Fanuc TP program (LS listing): FOLGE020.LS

/PROG  FOLGE020
/ATTR
OWNER		= GME;
COMMENT		= "VW336";
PROG_SIZE	= 7468;
CREATE		= DATE 16-09-30  TIME 23:12:18;
MODIFIED	= DATE 23-07-29  TIME 10:10:58;
FILE_NAME	= FOLGE020;
VERSION		= 0;
LINE_COUNT	= 47;
MEMORY_SIZE	= 11772;
PROTECT		= READ_WRITE;
TCD:  STACK_SIZE	= 500,
      TASK_PRIORITY	= 50,
      TIME_SLICE	= 0,
      BUSY_LAMP_OFF	= 0,
      ABORT_REQUEST	= 0,
      PAUSE_REQUEST	= 0;
DEFAULT_GROUP	= 1,1,1,1,*;
CONTROL_CODE	= 00000000 00000000;
/APPL
/MN
   1:  UFRAME_NUM=0 ;
   2:  UTOOL_NUM=1 ;
   3:  PAYLOAD[1] ;
   4:J P[1] 10% CNT0 ACC100 TB   0.00sec,P-SPS    ;
      1:  IF (DO[12]),CALL MAKRO998 ;
      2:  DO[15]=ON ;
      3:  DO[16]=ON ;
      4:  CALL MAKRO000    ;
      5:  WAIT (DI[9])    ;
       ------ ;
   5:  !Liberaciones PLC ;
   6:  !Fresado Estacionario SP1 ;
   7:  !Purgar KL1 ;
   8:J P[2] 100% CNT0 ACC100 TB   0.00sec,P-SPS    ;
      1:  TC_ONLINE (ON) ;
      4:  DO[23]=OFF ;
     32:  !Apagar Posicion base ;
     33:  DO[15]=OFF ;
      2:  !Espera fin de purga en casa ;
      3:  WAIT ((!DI[1534] AND !DI[1535]) OR !F[346] OR DI[15])    ;
      5:  TIMER[1]=RESET ;
      6:  TIMER[1]=START ;
      7:  CALL MAKRO050    ;
      8:  !Lib. Herramientas ;
      9:  DO[80]=ON ;
     10:  DO[79]=ON ;
     11:  DO[78]=OFF ;
     12:  DO[77]=OFF ;
     13:  DO[76]=ON ;
     14:  DO[75]=OFF ;
     15:  DO[74]=OFF ;
     16:  DO[73]=ON ;
     17:  DO[72]=ON ;
     18:  DO[71]=OFF ;
     19:  DO[70]=OFF ;
     20:  DO[69]=OFF ;
     21:  DO[68]=OFF ;
     22:  DO[67]=OFF ;
     23:  !Anticolisiones Robot ;
     24:  DO[41]=ON ;
     25:  DO[42]=ON ;
     26:  DO[43]=ON ;
     27:  DO[44]=ON ;
     28:  DO[53]=ON ;
     29:  DO[54]=ON ;
     30:  DO[55]=ON ;
     31:  DO[56]=ON ;
     34:  !Inicializar Garra ;
     35:  WAIT (M[2])    ;
     36:  F[1]=(ON) ;
     37:  F[2]=(ON) ;
     38:  F[3]=(ON) ;
     39:  F[4]=(ON) ;
     40:  F[5]=(ON) ;
     41:  IF (M[2]),CALL MAKRO342 ;
     42:  CALL MAKRO340    ;
     43:  WAIT (M[31] AND M[33] AND M[35] AND M[37] AND M[39])    ;
     44:  !Fresado SP1 ;
     45:  F[298]=(OFF) ;
     46:  CALL VW_USER(Basic1,EZSP,Nr1,ProgNr=31, , ,S-Punkt=31, ,EIN/AUS=ON) ;
     47:  WAIT    .10(sec) ;
     48:  F[79]=((DI[786] AND !DI[788]) OR (!DI[788] AND DI[130])) ;
     49:  F[78]=(DI[788] AND !F[79]) ;
     50:  GO[2]=(R[197]) ;
     51:  IF (F[78] AND F[79]),CALL MAKRO085 ;
     52:  IF (F[78] OR F[79]),CALL MAKRO084 ;
     53:  WAIT (M[96])    ;
     54:  !Seleccionar Pistola 1 ;
     55:  DO[1521]=ON ;
     56:  DO[1522]=OFF ;
     57:  DO[1523]=OFF ;
     58:  !Confirmacion Pistola 1 ;
     59:  WAIT (DI[1521] AND !DI[1522] AND !DI[1523])    ;
     60:  !Programa ;
     61:  GO[10]=(20) ;
     62:  !Parametro ;
     63:  GO[11]=(1) ;
     64:  WAIT    .10(sec) ;
     65:  !Purgar KL1 ;
     66:  IF (DI[1534] OR DI[163]),CALL MAKRO183 ;
     67:  WAIT (DI[23])    ;
     68:  DO[23]=ON ;
     69:  TC_ONLINE (M[2] AND M[30] AND M[31] AND M[33] AND M[35] AND M[37] AND M[39] AND M[95] AND M[96]) ;
       ------ ;
   9:  !Llamar a UP021 ;
  10:  !Tomar de la Estacion ST1350 ;
  11:  CALL UP021    ;
  12:  UFRAME_NUM=0 ;
  13:  UTOOL_NUM=1 ;
  14:J P[3] 100% CNT0 ACC100 TB    .10sec,P-SPS    ;
      1:  TC_ONLINE (ON) ;
      2:  DO[23]=OFF ;
      3:  WAIT (DI[23])    ;
      4:  DO[23]=ON ;
      5:  TC_ONLINE (M[3] AND M[30] AND M[31] AND M[34] AND M[35] AND M[37] AND M[39] AND M[95] AND M[96]) ;
       ------ ;
  15:  !Llamar a UP022 ;
  16:  !Tomar de la Estacion ST1360 ;
  17:  CALL UP022    ;
  18:  UFRAME_NUM=0 ;
  19:  UTOOL_NUM=1 ;
  20:J P[4] 100% CNT0 ACC100 TB    .10sec,P-SPS    ;
      1:  TC_ONLINE (ON) ;
      2:  DO[23]=OFF ;
      3:  WAIT (DI[23])    ;
      4:  DO[23]=ON ;
      5:  TC_ONLINE (M[1] AND M[30] AND M[31] AND M[34] AND M[36] AND M[38] AND M[39] AND M[95] AND M[96]) ;
       ------ ;
  21:  !Llamar a UP023 ;
  22:  !Soldadura ;
  23:  CALL UP023    ;
  24:  UFRAME_NUM=0 ;
  25:  UTOOL_NUM=1 ;
  26:J P[5] 100% CNT0 ACC100 TB    .10sec,P-SPS    ;
      1:  TC_ONLINE (ON) ;
      2:  DO[23]=OFF ;
      3:  !Fresado EZ1 ;
      4:  F[298]=(OFF) ;
      5:  CALL VW_USER(Basic1,EZSP,Nr1,ProgNr=31, , ,S-Punkt=31, ,EIN/AUS=ON) ;
      6:  WAIT    .10(sec) ;
      7:  F[79]=((DI[786] AND !DI[788]) OR (!DI[788] AND DI[130])) ;
      8:  F[78]=(DI[788] AND !F[79]) ;
      9:  GO[2]=(R[197]) ;
     10:  IF (F[78] OR F[79]),CALL MAKRO085 ;
     11:  IF (F[78] OR F[79]),CALL MAKRO084 ;
     12:  WAIT (M[96])    ;
     13:  WAIT (DI[23])    ;
     14:  DO[23]=ON ;
     15:  TC_ONLINE (M[1] AND M[30] AND M[31] AND M[34] AND M[36] AND M[38] AND M[39] AND M[95] AND M[96]) ;
       ------ ;
  27:  !Purgar ;
  28:  !UP024 Sello Estacionario ;
  29:  !UP070 Posicion Muestra ;
  30:  LBL[1] ;
  31:J P[6] 100% CNT0 ACC100 TB    .10sec,P-SPS    ;
      1:  TC_ONLINE (ON) ;
      2:  DO[23]=OFF ;
      3:  !Purgar KL1 ;
      4:  IF (DI[1534] OR DI[163]),CALL MAKRO183 ;
      5:  WAIT (DI[23])    ;
      6:  DO[23]=ON ;
      7:  TC_ONLINE (M[1] AND M[30] AND M[31] AND M[34] AND M[36] AND M[38] AND M[39] AND M[95] AND M[96]) ;
       ------ ;
  32:  CALL UP024    ;
  33:  IF (F[343] OR DI[162]),CALL UP070 ;
  34:  IF (F[343]),JMP LBL[1] ;
  35:  UFRAME_NUM=0 ;
  36:  UTOOL_NUM=1 ;
  37:  !En Area de Mantenimiento ;
  38:  !Llamar a UP025 ;
  39:  !Dejar en ST1380 ;
  40:J P[7] 100% CNT0 ACC100 TB    .10sec,P-SPS    ;
      1:  TC_ONLINE (ON) ;
      2:  DO[23]=OFF ;
      3:  LBL[1] ;
      4:  DO[18]=(ON) ;
      5:  WAIT ((DI[73] AND DI[72] AND !DI[60] AND DI[59] AND !DI[58] AND DI[57] AND !DI[18]) OR DI[19])    ;
      6:  IF (DI[19]),JMP LBL[3] ;
      7:  IF (DI[73] AND DI[72] AND !DI[60] AND DI[59] AND !DI[58] AND DI[57]),JMP LBL[2] ;
      8:  LBL[3] ;
      9:  IF (F[78] OR F[79]),CALL MAKRO084 ;
     10:  CALL MAKRO089    ;
     11:  DO[17]=(ON) ;
     12:  GO[19]=(11) ;
     13:  F[281]=(ON) ;
     14:  WAIT (DI[17])    ;
     15:  F[64]=(ON) ;
     16:  F[65]=(OFF) ;
     17:  F[66]=(OFF) ;
     18:  F[67]=(OFF) ;
     19:  LBL[4] ;
     20:  IF (DI[132] AND !DI[133] AND !DI[134] AND !DI[135] AND DI[17]),CALL MAKRO081 ;
     21:  IF (F[85]),JMP LBL[4] ;
     22:  CALL VW_USER(Basic1,EZSP,Nr1 Service,ProgNr=31, , ,S-Punkt=31, ,EIN/AUS=1) ;
     23:  F[79]=((!DI[788] AND DI[130]) OR (DI[786] AND !DI[788])) ;
     24:  F[78]=(DI[788] AND !F[79]) ;
     25:  GO[2]=(R[197]) ;
     26:  IF (F[78] OR F[79]),CALL MAKRO085 ;
     27:  IF (F[78] OR F[79]),CALL MAKRO084 ;
     28:  WAIT (M[96] AND !DI[132])    ;
     29:  DO[17]=(OFF) ;
     30:  GO[19]=(0) ;
     31:  WAIT (!DI[19])    ;
     32:  JMP LBL[1] ;
     33:  LBL[2] ;
     34:  DO[18]=(OFF) ;
     35:  F[281]=(OFF) ;
     36:  WAIT (DI[23])    ;
     37:  DO[23]=ON ;
     38:  TC_ONLINE (M[1] AND M[30] AND M[31] AND M[34] AND M[36] AND M[38] AND M[39] AND M[95] AND M[96]) ;
       ------ ;
  41:  CALL UP025    ;
  42:  UFRAME_NUM=0 ;
  43:  UTOOL_NUM=1 ;
  44:J P[8] 100% CNT0 ACC100 TB    .10sec,P-SPS    ;
      1:  TC_ONLINE (ON) ;
      2:  DO[23]=OFF ;
      3:  F[298]=(OFF) ;
      4:  CALL VW_USER(Basic1,EZSP,Nr1,ProgNr=31, , ,S-Punkt=31, ,EIN/AUS=ON) ;
      5:  WAIT    .10(sec) ;
      6:  F[79]=((DI[786] AND !DI[788]) OR (!DI[788] AND DI[130])) ;
      7:  F[78]=(DI[788] AND !F[79]) ;
      8:  GO[2]=(R[197]) ;
      9:  IF (F[78] AND F[79]),CALL MAKRO085 ;
     10:  IF (F[78] OR F[79]),CALL MAKRO084 ;
     11:  WAIT (M[96])    ;
     12:  WAIT (DI[23])    ;
     13:  DO[23]=ON ;
     14:  TC_ONLINE (M[2] AND M[30] AND M[31] AND M[33] AND M[35] AND M[37] AND M[39] AND M[95] AND M[96]) ;
       ------ ;
  45:  !Fin de Trabajo Total ;
  46:J P[9] 100% CNT0 ACC100 TB    .10sec,P-SPS    ;
      1:  TC_ONLINE (ON) ;
      2:  DO[23]=OFF ;
      3:  CALL MAKRO015    ;
      4:  WAIT (DI[23])    ;
      5:  DO[23]=ON ;
      6:  TC_ONLINE (M[2] AND M[30] AND M[31] AND M[33] AND M[35] AND M[37] AND M[39] AND M[95] AND M[96]) ;
       ------ ;
  47:J P[10] 100% CNT0 ACC100 TB   0.00sec,P-SPS    ;
      1:  TC_ONLINE (ON) ;
      2:  DO[14]=ON ;
      3:  DO[15]=ON ;
      4:  TIMER[1]=STOP ;
      5:  TIMER[2]=(TIMER[1]) ;
      6:  TIMER[2]=STOP ;
       ------ ;
/POS
P[1]{
   GP1:
	UF : 0, UT : 1,		CONFIG : 'N U T, 0, 0, -1',
	X =  1190.730  mm,	Y =  -289.205  mm,	Z =  1231.849  mm,
	W =   -30.000 deg,	P =     0.000 deg,	R =    30.000 deg
   GP2:
	UF : 0, UT : 1,
	J1=   100.000  mm
   GP3:
	UF : 0, UT : 1,
	J1=     0.000  mm
   GP4:
	UF : 0, UT : 1,
	J1=     0.000  mm
};
P[2]{
   GP1:
	UF : 0, UT : 1,		CONFIG : 'N U T, 0, 0, -1',
	X =  1190.730  mm,	Y =  -289.205  mm,	Z =  1231.849  mm,
	W =   -30.000 deg,	P =     0.000 deg,	R =    30.000 deg
   GP2:
	UF : 0, UT : 1,
	J1=   100.000  mm
   GP3:
	UF : 0, UT : 1,
	J1=     0.000  mm
   GP4:
	UF : 0, UT : 1,
	J1=     0.000  mm
};
P[3]{
   GP1:
	UF : 0, UT : 1,		CONFIG : 'N U T, 0, 0, -1',
	X =  1190.730  mm,	Y =  -289.205  mm,	Z =  1231.849  mm,
	W =   -30.000 deg,	P =     0.000 deg,	R =    30.000 deg
   GP2:
	UF : 0, UT : 1,
	J1=   100.000  mm
   GP3:
	UF : 0, UT : 1,
	J1=     0.000  mm
   GP4:
	UF : 0, UT : 1,
	J1=     0.000  mm
};
P[4]{
   GP1:
	UF : 0, UT : 1,		CONFIG : 'N U T, 0, 0, -1',
	X =  1190.730  mm,	Y =  -289.205  mm,	Z =  1231.849  mm,
	W =   -30.000 deg,	P =     0.000 deg,	R =    30.000 deg
   GP2:
	UF : 0, UT : 1,
	J1=   100.000  mm
   GP3:
	UF : 0, UT : 1,
	J1=     0.000  mm
   GP4:
	UF : 0, UT : 1,
	J1=     0.000  mm
};
P[5]{
   GP1:
	UF : 0, UT : 1,		CONFIG : 'N U T, 0, 0, -1',
	X =  1190.730  mm,	Y =  -289.205  mm,	Z =  1231.849  mm,
	W =   -30.000 deg,	P =     0.000 deg,	R =    30.000 deg
   GP2:
	UF : 0, UT : 1,
	J1=   100.000  mm
   GP3:
	UF : 0, UT : 1,
	J1=     0.000  mm
   GP4:
	UF : 0, UT : 1,
	J1=     0.000  mm
};
P[6]{
   GP1:
	UF : 0, UT : 1,		CONFIG : 'N U T, 0, 0, -1',
	X =  1190.730  mm,	Y =  -289.205  mm,	Z =  1231.849  mm,
	W =   -30.000 deg,	P =     0.000 deg,	R =    30.000 deg
   GP2:
	UF : 0, UT : 1,
	J1=   100.000  mm
   GP3:
	UF : 0, UT : 1,
	J1=     0.000  mm
   GP4:
	UF : 0, UT : 1,
	J1=     0.000  mm
};
P[7]{
   GP1:
	UF : 0, UT : 1,		CONFIG : 'N U T, 0, 0, -1',
	X =  1190.730  mm,	Y =  -289.205  mm,	Z =  1231.849  mm,
	W =   -30.000 deg,	P =     0.000 deg,	R =    30.000 deg
   GP2:
	UF : 0, UT : 1,
	J1=   100.000  mm
   GP3:
	UF : 0, UT : 1,
	J1=     0.000  mm
   GP4:
	UF : 0, UT : 1,
	J1=     0.000  mm
};
P[8]{
   GP1:
	UF : 0, UT : 1,		CONFIG : 'N U T, 0, 0, -1',
	X =  1190.730  mm,	Y =  -289.205  mm,	Z =  1231.849  mm,
	W =   -30.000 deg,	P =     0.000 deg,	R =    30.000 deg
   GP2:
	UF : 0, UT : 1,
	J1=   100.000  mm
   GP3:
	UF : 0, UT : 1,
	J1=     0.000  mm
   GP4:
	UF : 0, UT : 1,
	J1=     0.000  mm
};
P[9]{
   GP1:
	UF : 0, UT : 1,		CONFIG : 'N U T, 0, 0, -1',
	X =  1190.730  mm,	Y =  -289.205  mm,	Z =  1231.849  mm,
	W =   -30.000 deg,	P =     0.000 deg,	R =    30.000 deg
   GP2:
	UF : 0, UT : 1,
	J1=   100.000  mm
   GP3:
	UF : 0, UT : 1,
	J1=     0.000  mm
   GP4:
	UF : 0, UT : 1,
	J1=     0.000  mm
};
P[10]{
   GP1:
	UF : 0, UT : 1,		CONFIG : 'N U T, 0, 0, -1',
	X =  1190.730  mm,	Y =  -289.205  mm,	Z =  1231.849  mm,
	W =   -30.000 deg,	P =     0.000 deg,	R =    30.000 deg
   GP2:
	UF : 0, UT : 1,
	J1=   100.000  mm
   GP3:
	UF : 0, UT : 1,
	J1=     0.000  mm
   GP4:
	UF : 0, UT : 1,
	J1=     0.000  mm
};
/END
